Fanuc KAREL source: ka00195.KL

-- PROVISIONAL review KL for V940-1; original PC SHA256 63d8ed4802aa1d4efa53768760aedbd46227d824fddfd43c6a3a89be3f177636
-- Incomplete behavior may be omitted. Consult companion uncertainty JSON. Do not deploy.
PROGRAM KA00195
%NOLOCKGROUP
-- UNRESOLVED_DECL SRC type=002017
-- UNRESOLVED_DECL DST type=002017
BEGIN
  -- V9_COMPOSED_GLOBAL_TRANSFER_HINT repetitions=1; address IDs observed; pairing/direction/source/runtime held
  -- V9_TWO_GLOBAL_ADDRESS_COPY_HINT bounded five-record physical form; type/direction/source/runtime held
  -- V9_ZERO_TABLE_METADATA_HINT layout=0001; no indexed target words; source/name/runtime held
  -- UNRESOLVED_PC offsets 5-19; opcodes 22,22,1E
  -- UNRESOLVED_PC offsets 24-28; opcodes 7F
END KA00195
